INTERFACE I_Observable EXTENDS I_Object

METHOD Attach : BOOL
VAR_INPUT
    ipObserver:         I_Observer;
END_VAR
END_METHOD

(*Notify automatically on write access of observable value*)
PROPERTY bAutoNotify : BOOL
GET
END_GET
SET
END_SET
END_PROPERTY

(*Notify only when the value is actually changed*)
PROPERTY bNotifyWhenChanged : BOOL
GET
END_GET
SET
END_SET
END_PROPERTY

METHOD Detach : BOOL
VAR_INPUT
    ipObserver:         I_Observer;
END_VAR
END_METHOD

PROPERTY nDataSize : UDINT
GET
END_GET
END_PROPERTY

PROPERTY nObserverCount : UDINT
GET
END_GET
END_PROPERTY

METHOD NotifyAll : I_Observable
VAR_INPUT
END_VAR
END_METHOD

METHOD NotifyLast : I_Observable
VAR_INPUT
END_VAR
END_METHOD

PROPERTY nTypeClass : __SYSTEM.TYPE_CLASS
GET
END_GET
END_PROPERTY

METHOD ABSTRACT ValueChanged : BOOL
VAR_INPUT
END_VAR
END_METHOD

END_INTERFACE

(* stored: Version 1.1.0.1, ProductVersion 3.1.4024.12
   Itf I_Observable: Id {e9d5ee08-eb7e-494a-b197-8f922f772785}
   Method Attach: Id {30211a61-21d5-40ca-8122-c8c8f2acdb97}
   Property bAutoNotify: Id {b2bbc409-bd98-0bad-2172-8600de7556d9}
   Get Get: Id {28c68bd4-00ea-01a3-1246-c18fa2952457}
   Set Set: Id {868424c9-4d32-097c-04cf-be577c5a0bca}
   Property bNotifyWhenChanged: Id {dba79f02-ec11-0ccb-0ffe-bd21359f971e}
   Get Get: Id {111601c9-958a-0fcb-2da5-91de6c92f0b8}
   Set Set: Id {c362826d-df63-0759-2036-76c0288d7680}
   Method Detach: Id {ebccaf28-c550-4b56-881b-b9dc49898d61}
   Property nDataSize: Id {66ccf410-7b87-46bb-a40d-a3f511a75616}
   Get Get: Id {a9718243-75e3-46d3-8875-a897e41ceb90}
   Property nObserverCount: Id {07d52f56-10f6-4076-aab3-6b8ebc9310fa}
   Get Get: Id {3a19d823-a61c-41a4-83cb-832f68ece898}
   Method NotifyAll: Id {dca0986e-fc2a-4198-a535-6eefd7c6a6f6}
   Method NotifyLast: Id {269f7bdd-fe70-43f6-bffb-4ca342e2c104}
   Property nTypeClass: Id {cf93b4e0-71b2-07a5-03a3-df12d61358cf}
   Get Get: Id {fc7fe750-ffac-0880-2964-730a12b0f2e2}
   Method ValueChanged: Id {fe01f384-fa15-0491-29cb-2dd7249fb59a} *)
